PROGRAM Move_Vel
VAR
	MC_MoveVelocity5: MC_MoveVelocity;
	MC_MoveVelocity6: MC_MoveVelocity;
END_VAR


AXIS();

MC_MoveVelocity5(
	Axis:= AXIS.Axis5, 
	Execute:= , 
	Velocity:= MAIN.VEL_REQ1.VEL5, 
	Acceleration:= , 
	Deceleration:= , 
	Jerk:= , 
	Direction:= , 
	BufferMode:= , 
	Options:= , 
	InVelocity=> , 
	Busy=> , 
	Active=> , 
	CommandAborted=> , 
	Error=> , 
	ErrorID=> );
MC_MoveVelocity6(
	Axis:= AXIS.Axis6, 
	Execute:= , 
	Velocity:= MAIN.VEL_REQ1.VEL6, 
	Acceleration:= , 
	Deceleration:= , 
	Jerk:= , 
	Direction:= , 
	BufferMode:= , 
	Options:= , 
	InVelocity=> , 
	Busy=> , 
	Active=> , 
	CommandAborted=> , 
	Error=> , 
	ErrorID=> );

END_PROGRAM

(* stored: Version 1.1.0.1, ProductVersion 3.1.4024.0
   POU Move_Vel: Id {e60ff0ff-b7cb-4aa6-9273-e830ad3f72fc}, SpecialFunc None *)
